FUNCTION F_ServoCheckWindow : BOOL
VAR_INPUT
	Unwind			: LREAL;
	Value			: LREAL;
	Target			: REAL;
	Tollerance		: REAL;
END_VAR
VAR
	UpperBound		: REAL;
	LowerBound		: REAL;
END_VAR

LowerBound := Target - Tollerance;
UpperBound := Target + Tollerance;

IF LowerBound >= 0 AND UpperBound <= Unwind THEN
	F_ServoCheckWindow := ((Value >= LowerBound) AND (Value <= UpperBound));
ELSIF LowerBound < 0 THEN
	F_ServoCheckWindow := (((Value >= (Unwind + LowerBound)) AND (Value <= Unwind)) OR (Value >= 0) AND (Value <= UpperBound));
ELSIF UpperBound > Unwind THEN
	F_ServoCheckWindow := (((Value >= LowerBound) AND (Value <= Unwind)) OR (Value >= 0) AND (Value <= (UpperBound - Unwind)));
ELSE
	F_ServoCheckWindow := FALSE;
END_IF

END_FUNCTION

(* stored: Version 1.1.0.1, ProductVersion 3.1.4024.3
   POU F_ServoCheckWindow: Id {a7e11f2e-404d-471f-bb43-752f5b8ec244}, SpecialFunc None *)
